(* IEC 61131-3 sources: openPLC_watertank/, 3 files *)

(* ---- original.st ---- *)
PROGRAM LatchLogic
VAR
    PB1      AT %QX100.0 : BOOL;   (* Start button  - Modbus coil 801 *)
    PB2      AT %QX100.1 : BOOL;   (* Stop button   - Modbus coil 802 *)
    PUMP     AT %QX0.0   : BOOL;   (* Pump output   - Modbus coil 1   *)
    TANK_FULL AT %QX100.2 : BOOL;  (* Tank Full Status - Modbus coil 803 *)
END_VAR

(* Start/Stop latch with Tank Full condition:
   - Press PB1 once to start (latches ON) unless Tank_Full is true
   - Press PB2 to stop (unlatch)
   - If Tank_Full becomes TRUE, the pump must stop immediately
   - The pump cannot start if Tank_Full is TRUE *)

(* Pump Control Logic *)
IF NOT TANK_FULL THEN
    (* Tank is not full, normal start/stop behavior *)
    IF PB1 THEN
        PUMP := TRUE;  (* Start pump *)
    END_IF;

    IF PB2 THEN
        PUMP := FALSE; (* Stop pump *)
    END_IF;
ELSE
    (* Tank is full, stop pump and prevent starting *)
    PUMP := FALSE;  (* Ensure pump is OFF *)
END_IF;

END_PROGRAM

CONFIGURATION Config0
   RESOURCE Res0 ON PLC
      TASK task0(INTERVAL := T#100ms, PRIORITY := 0);
      PROGRAM instance0 WITH task0 : LatchLogic;
   END_RESOURCE
END_CONFIGURATION

(* ---- tank2.st ---- *)
PROGRAM LatchLogic
VAR
    PB1      AT %QX100.0 : BOOL;   (* Start button  - Modbus coil 801 *)
    PB2      AT %QX100.1 : BOOL;   (* Stop button   - Modbus coil 802 *)
    PUMP     AT %QX0.0   : BOOL;   (* Pump output   - Modbus coil 1   *)
    TANK_FULL AT %QX100.2 : BOOL;  (* Tank Full Status - Modbus coil 803 *)
    Tank_Level AT %QW0 : INT;      (* Tank level 0-100% - Modbus holding reg 40001 *)
END_VAR

(* Start/Stop latch with Tank Full condition:
   - Press PB1 once to start (latches ON) unless Tank_Full is true
   - Press PB2 to stop (unlatch)
   - If Tank_Full becomes TRUE, the pump must stop immediately
   - The pump cannot start if Tank_Full is TRUE *)

(* Pump Control Logic *)
IF NOT TANK_FULL THEN
    (* Tank is not full, normal start/stop behavior *)
    IF PB1 THEN
        PUMP := TRUE;  (* Start pump *)
    END_IF;

    IF PB2 THEN
        PUMP := FALSE; (* Stop pump *)
    END_IF;
ELSE
    (* Tank is full, stop pump and prevent starting *)
    PUMP := FALSE;  (* Ensure pump is OFF *)
END_IF;

END_PROGRAM

CONFIGURATION Config0
   RESOURCE Res0 ON PLC
      TASK task0(INTERVAL := T#100ms, PRIORITY := 0);
      PROGRAM instance0 WITH task0 : LatchLogic;
   END_RESOURCE
END_CONFIGURATION

(* ---- WaterTankPump.st ---- *)
PROGRAM WaterTankPump
VAR
    PB_Start  AT %QX100.0 : BOOL;   (* Start button - Modbus coil 801 *)
    PB_Stop   AT %QX100.1 : BOOL;   (* Stop button - Modbus coil 802 *)
    Tank_Full AT %QX100.3 : BOOL;   (* Tank full sensor - Modbus coil 803 *)
    Tank_Level AT %QW100 : INT;     (* Tank level - Modbus holding reg 40001 *)
    Pump_Motor AT %QX0.0 : BOOL;    (* Pump output - Modbus coil 1 *)
    Pump_Run : BOOL;                (* Internal latch state *)
END_VAR

(* Normal latch logic: start/stop *)
IF PB_Start AND NOT Tank_Full THEN
    Pump_Run := TRUE;
END_IF;

IF PB_Stop THEN
    Pump_Run := FALSE;
END_IF;

(* Emergency override *)
IF Tank_Full THEN
    Pump_Run := FALSE;
END_IF;

(* Drive motor output *)
Pump_Motor := Pump_Run;

END_PROGRAM

CONFIGURATION Config0
   RESOURCE Res0 ON PLC
      TASK task0(INTERVAL := T#100ms, PRIORITY := 0);
      PROGRAM instance0 WITH task0 : WaterTankPump;
   END_RESOURCE
END_CONFIGURATION
